% RSLogix 500 project P8_BAK007.RSS, saved by version 12.00.00.00 %
PROJECT "UNTITLED"    % processor: Bul.1763 MicroLogix 1100 Series B %

PROGRAM FILES
  LAD 2   5 rungs

DATA FILES
  O0 OUTPUT  4 elements
  I1 INPUT  6 elements
  S2 STATUS  66 elements
  B3 BINARY  1 elements
  T4 TIMER  1 elements
  C5 COUNTER  1 elements
  R6 CONTROL  1 elements
  N7 INTEGER  6 elements
  F8 FLOAT  3 elements

LADDER 2
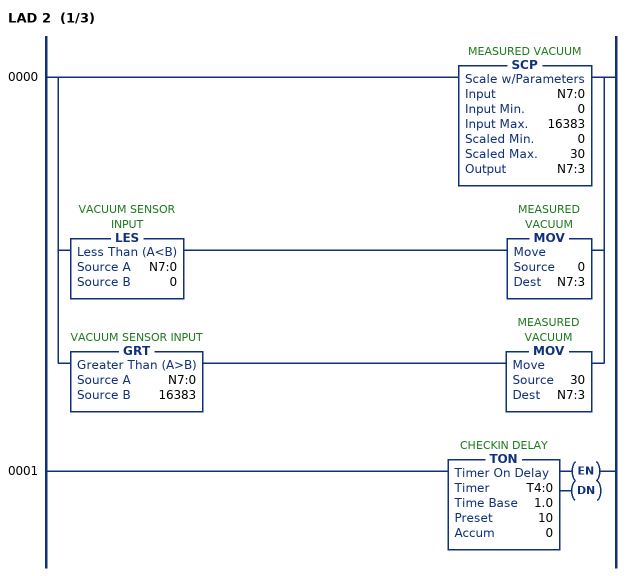
% Rung: 0 %
SOR BST SCP N7:0 0 16383 0 30 N7:3 NXB LES N7:0 0 MOV 0 N7:3 NXB GRT N7:0 16383 MOV 30 N7:3 BND EOR
%   N7:0  "VACUUM SENSOR INPUT" %
%   N7:3  "MEASURED VACUUM" %
% Rung: 1 %
SOR TON T4:0 1.0 10 0 EOR
%   T4:0  "CHECKIN DELAY" %

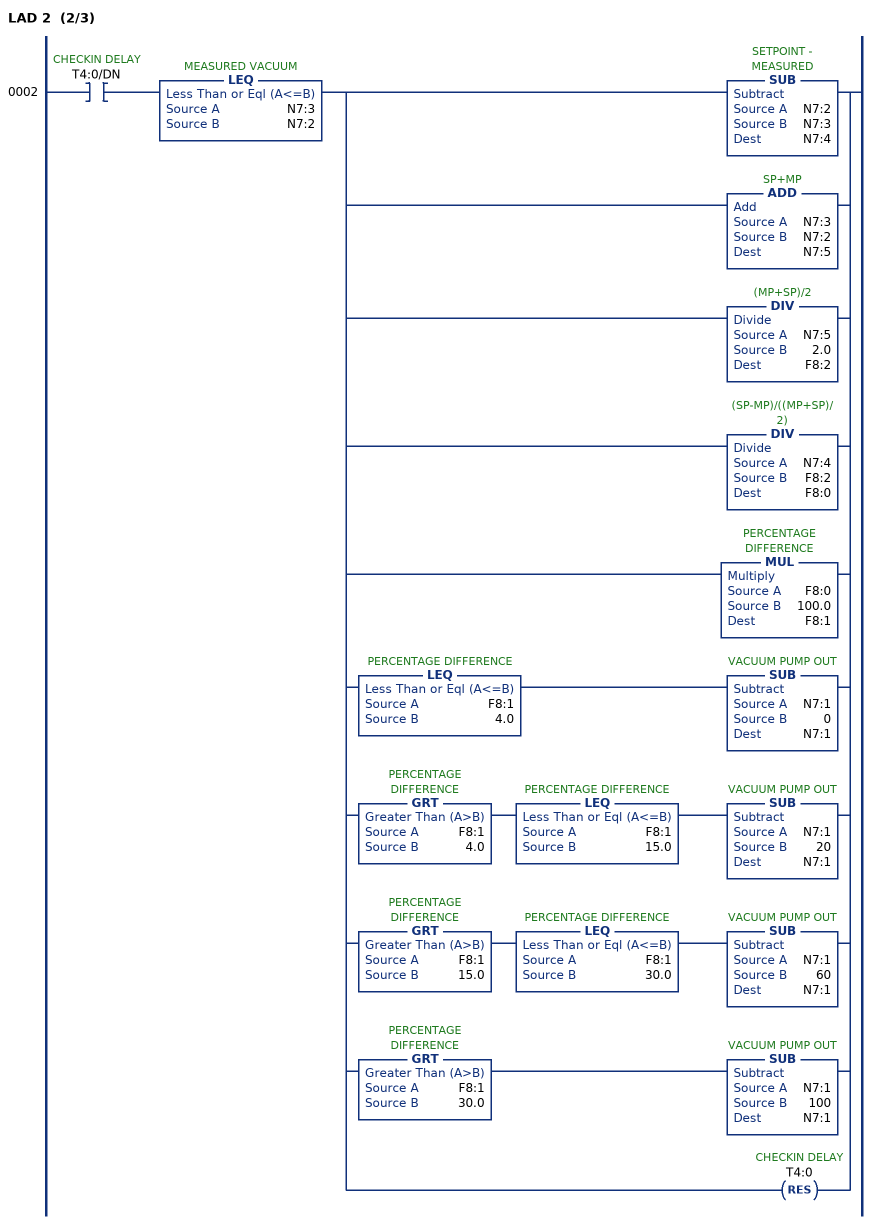
% Rung: 2 %
SOR XIC T4:0/DN LEQ N7:3 N7:2 BST SUB N7:2 N7:3 N7:4 NXB ADD N7:3 N7:2 N7:5 NXB DIV N7:5 2.0 F8:2 NXB DIV N7:4 F8:2 F8:0 NXB MUL F8:0 100.0 F8:1 NXB LEQ F8:1 4.0 SUB N7:1 0 N7:1 NXB GRT F8:1 4.0 LEQ F8:1 15.0 SUB N7:1 20 N7:1 NXB GRT F8:1 15.0 LEQ F8:1 30.0 SUB N7:1 60 N7:1 NXB GRT F8:1 30.0 SUB N7:1 100 N7:1 NXB RES T4:0 BND EOR
%   T4:0  "CHECKIN DELAY" %
%   N7:3  "MEASURED VACUUM" %
%   N7:2  "VACUUM SETPOINT" %
%   N7:4  "SETPOINT - MEASURED" %
%   N7:5  "SP+MP" %
%   F8:2  "(MP+SP)/2" %
%   F8:0  "(SP-MP)/((MP+SP)/2)" %
%   F8:1  "PERCENTAGE DIFFERENCE" %
%   N7:1  "VACUUM PUMP OUT" %

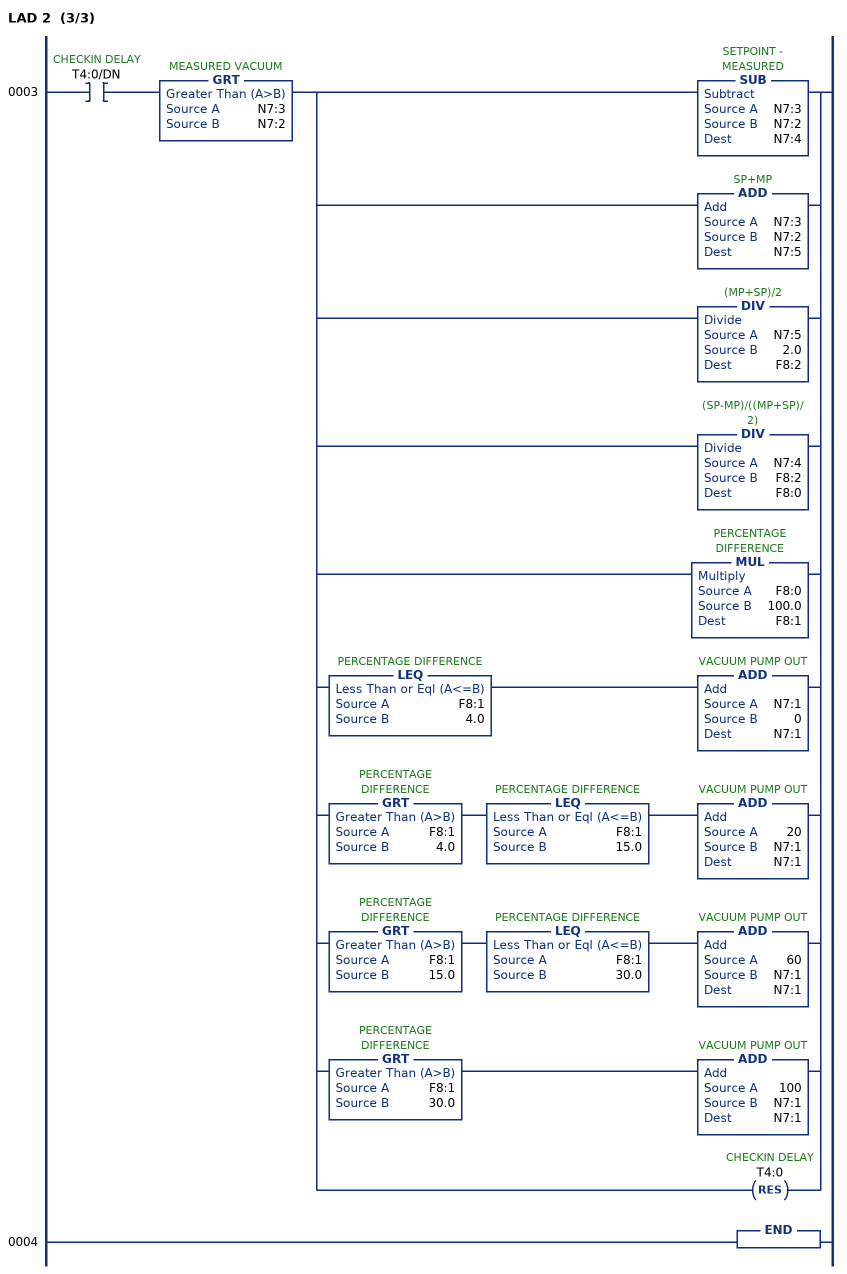
% Rung: 3 %
SOR XIC T4:0/DN GRT N7:3 N7:2 BST SUB N7:3 N7:2 N7:4 NXB ADD N7:3 N7:2 N7:5 NXB DIV N7:5 2.0 F8:2 NXB DIV N7:4 F8:2 F8:0 NXB MUL F8:0 100.0 F8:1 NXB LEQ F8:1 4.0 ADD N7:1 0 N7:1 NXB GRT F8:1 4.0 LEQ F8:1 15.0 ADD 20 N7:1 N7:1 NXB GRT F8:1 15.0 LEQ F8:1 30.0 ADD 60 N7:1 N7:1 NXB GRT F8:1 30.0 ADD 100 N7:1 N7:1 NXB RES T4:0 BND EOR
%   T4:0  "CHECKIN DELAY" %
%   N7:3  "MEASURED VACUUM" %
%   N7:2  "VACUUM SETPOINT" %
%   N7:4  "SETPOINT - MEASURED" %
%   N7:5  "SP+MP" %
%   F8:2  "(MP+SP)/2" %
%   F8:0  "(SP-MP)/((MP+SP)/2)" %
%   F8:1  "PERCENTAGE DIFFERENCE" %
%   N7:1  "VACUUM PUMP OUT" %
% Rung: 4 %
SOR END EOR

DATA TABLE (non-zero values as saved)
DATA T4
% .PRE .ACC %
% T4:0 % 10 0
DATA F8
% F8:0 % 0.06896552 6.896552 14.5
